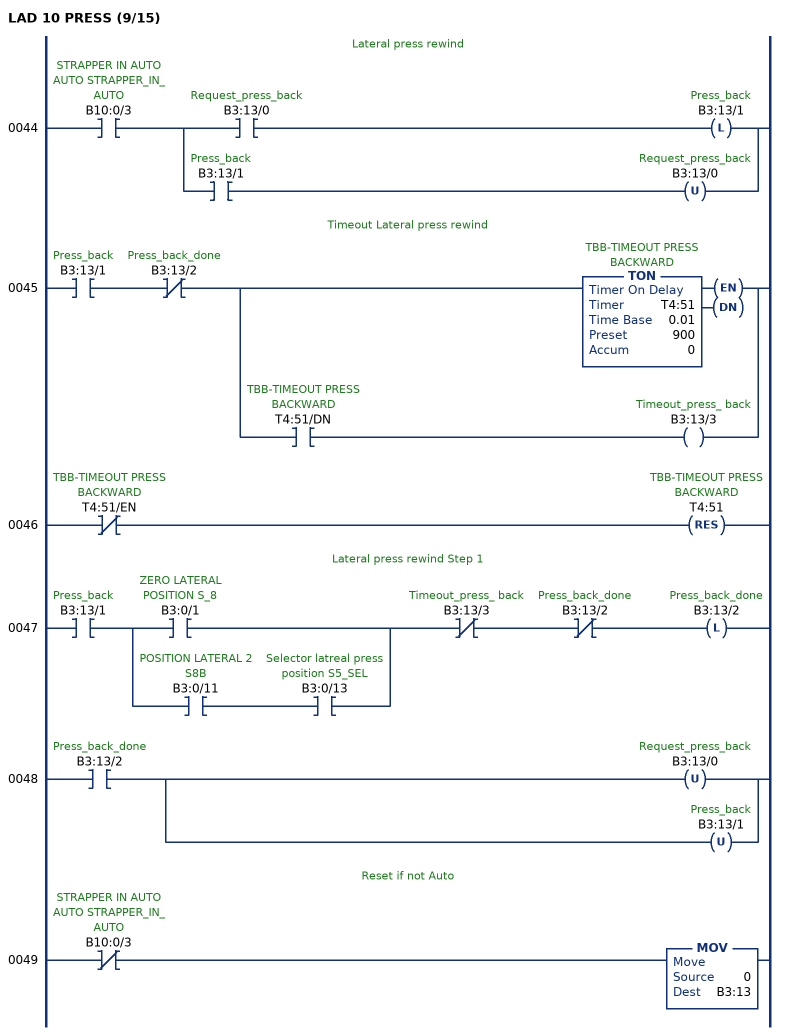
% Rung: 44 %
% Lateral press rewind %
SOR XIC B10:0/3 BST XIC B3:13/0 OTL B3:13/1 NXB XIC B3:13/1 OTU B3:13/0 BND EOR
%   B10:0/3  STRAPPER_IN_AUTO  "STRAPPER IN AUTO AUTO" %
%   B3:13/0  "Request_press_back" %
%   B3:13/1  "Press_back" %
% Rung: 45 %
% Timeout Lateral press rewind %
SOR XIC B3:13/1 XIO B3:13/2 BST TON T4:51 0.01 900 0 NXB XIC T4:51/DN OTE B3:13/3 BND EOR
%   B3:13/1  "Press_back" %
%   B3:13/2  "Press_back_done" %
%   T4:51  "TBB-TIMEOUT PRESS BACKWARD" %
%   B3:13/3  "Timeout_press_ back" %
% Rung: 46 %
SOR XIO T4:51/EN RES T4:51 EOR
%   T4:51  "TBB-TIMEOUT PRESS BACKWARD" %
% Rung: 47 %
% Lateral press rewind Step 1 %
SOR XIC B3:13/1 BST XIC B3:0/1 NXB XIC B3:0/11 XIC B3:0/13 BND XIO B3:13/3 XIO B3:13/2 OTL B3:13/2 EOR
%   B3:13/1  "Press_back" %
%   B3:0/1  S_8  "ZERO LATERAL POSITION" %
%   B3:0/11  S8B  "POSITION LATERAL 2" %
%   B3:0/13  S5_SEL  "Selector latreal press position" %
%   B3:13/3  "Timeout_press_ back" %
%   B3:13/2  "Press_back_done" %
% Rung: 48 %
SOR XIC B3:13/2 BST OTU B3:13/0 NXB OTU B3:13/1 BND EOR
%   B3:13/2  "Press_back_done" %
%   B3:13/0  "Request_press_back" %
%   B3:13/1  "Press_back" %
% Rung: 49 %
% Reset if not Auto %
SOR XIO B10:0/3 MOV 0 B3:13 EOR
%   B10:0/3  STRAPPER_IN_AUTO  "STRAPPER IN AUTO AUTO" %

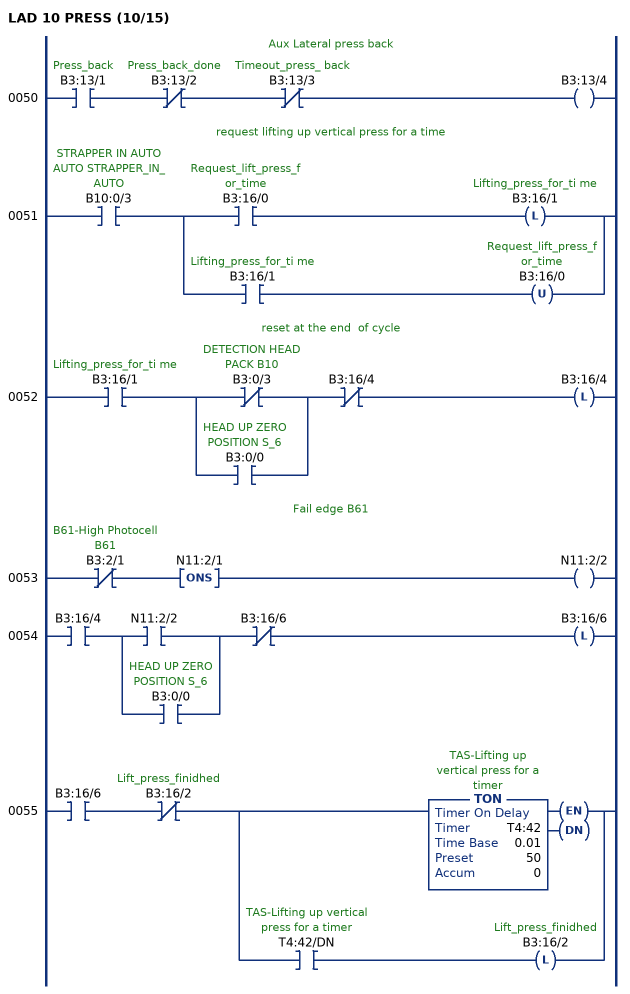
% Rung: 50 %
% Aux Lateral press back %
SOR XIC B3:13/1 XIO B3:13/2 XIO B3:13/3 OTE B3:13/4 EOR
%   B3:13/1  "Press_back" %
%   B3:13/2  "Press_back_done" %
%   B3:13/3  "Timeout_press_ back" %
% Rung: 51 %
% request lifting up vertical press for a time %
SOR XIC B10:0/3 BST XIC B3:16/0 OTL B3:16/1 NXB XIC B3:16/1 OTU B3:16/0 BND EOR
%   B10:0/3  STRAPPER_IN_AUTO  "STRAPPER IN AUTO AUTO" %
%   B3:16/0  "Request_lift_press_f or_time" %
%   B3:16/1  "Lifting_press_for_ti me" %
% Rung: 52 %
% reset at the end  of cycle %
SOR XIC B3:16/1 BST XIO B3:0/3 NXB XIC B3:0/0 BND XIO B3:16/4 OTL B3:16/4 EOR
%   B3:16/1  "Lifting_press_for_ti me" %
%   B3:0/3  B10  "DETECTION HEAD PACK" %
%   B3:0/0  S_6  "HEAD UP ZERO POSITION" %
% Rung: 53 %
% Fail edge B61 %
SOR XIO B3:2/1 ONS N11:2/1 OTE N11:2/2 EOR
%   B3:2/1  B61  "B61-High Photocell" %
% Rung: 54 %
SOR XIC B3:16/4 BST XIC N11:2/2 NXB XIC B3:0/0 BND XIO B3:16/6 OTL B3:16/6 EOR
%   B3:0/0  S_6  "HEAD UP ZERO POSITION" %
% Rung: 55 %
SOR XIC B3:16/6 XIO B3:16/2 BST TON T4:42 0.01 50 0 NXB XIC T4:42/DN OTL B3:16/2 BND EOR
%   B3:16/2  "Lift_press_finidhed" %
%   T4:42  "TAS-Lifting up vertical press for a timer" %

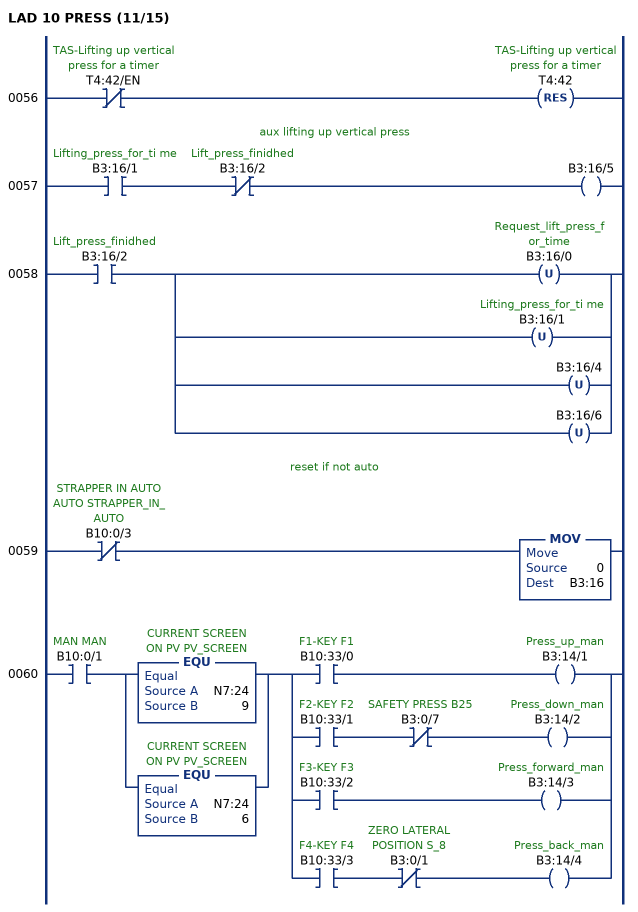
% Rung: 56 %
SOR XIO T4:42/EN RES T4:42 EOR
%   T4:42  "TAS-Lifting up vertical press for a timer" %
% Rung: 57 %
% aux lifting up vertical press %
SOR XIC B3:16/1 XIO B3:16/2 OTE B3:16/5 EOR
%   B3:16/1  "Lifting_press_for_ti me" %
%   B3:16/2  "Lift_press_finidhed" %
% Rung: 58 %
SOR XIC B3:16/2 BST OTU B3:16/0 NXB BST OTU B3:16/1 NXB BST OTU B3:16/4 NXB OTU B3:16/6 BND BND BND EOR
%   B3:16/2  "Lift_press_finidhed" %
%   B3:16/0  "Request_lift_press_f or_time" %
%   B3:16/1  "Lifting_press_for_ti me" %
% Rung: 59 %
% reset if not auto %
SOR XIO B10:0/3 MOV 0 B3:16 EOR
%   B10:0/3  STRAPPER_IN_AUTO  "STRAPPER IN AUTO AUTO" %
% Rung: 60 %
SOR XIC B10:0/1 BST EQU N7:24 9 NXB EQU N7:24 6 BND BST XIC B10:33/0 OTE B3:14/1 NXB BST XIC B10:33/1 XIO B3:0/7 OTE B3:14/2 NXB BST XIC B10:33/2 OTE B3:14/3 NXB XIC B10:33/3 XIO B3:0/1 OTE B3:14/4 BND BND BND EOR
%   B10:0/1  MAN  "MAN" %
%   N7:24  PV_SCREEN  "CURRENT SCREEN ON PV" %
%   B10:33/0  F1  "F1-KEY" %
%   B3:14/1  "Press_up_man" %
%   B10:33/1  F2  "F2-KEY" %
%   B3:0/7  B25  "SAFETY PRESS" %
%   B3:14/2  "Press_down_man" %
%   B10:33/2  F3  "F3-KEY" %
%   B3:14/3  "Press_forward_man" %
%   B10:33/3  F4  "F4-KEY" %
%   B3:0/1  S_8  "ZERO LATERAL POSITION" %
%   B3:14/4  "Press_back_man" %

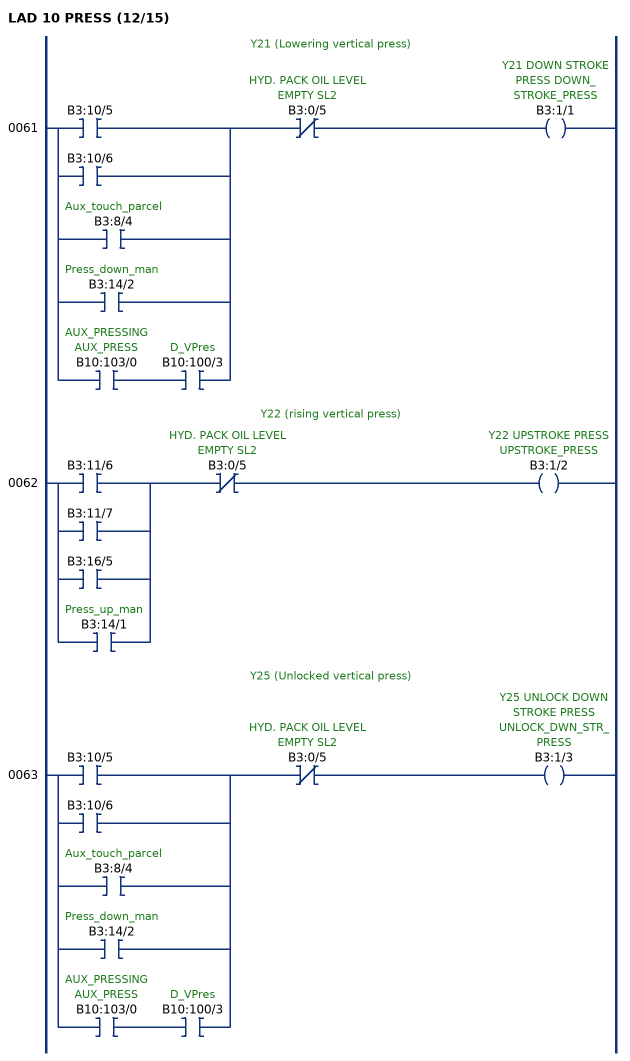
% Rung: 61 %
% Y21 (Lowering vertical press) %
SOR BST BST BST XIC B3:10/5 NXB BST XIC B3:10/6 NXB XIC B3:8/4 BND BND NXB XIC B3:14/2 BND NXB XIC B10:103/0 XIC B10:100/3 BND XIO B3:0/5 OTE B3:1/1 EOR
%   B3:8/4  "Aux_touch_parcel" %
%   B3:14/2  "Press_down_man" %
%   B10:103/0  AUX_PRESS  "AUX_PRESSING" %
%   B10:100/3  "D_VPres" %
%   B3:0/5  SL2  "HYD. PACK OIL LEVEL EMPTY" %
%   B3:1/1  DOWN_STROKE_PRESS  "Y21 DOWN STROKE PRESS" %
% Rung: 62 %
% Y22 (rising vertical press) %
SOR BST BST XIC B3:11/6 NXB BST XIC B3:11/7 NXB XIC B3:16/5 BND BND NXB XIC B3:14/1 BND XIO B3:0/5 OTE B3:1/2 EOR
%   B3:14/1  "Press_up_man" %
%   B3:0/5  SL2  "HYD. PACK OIL LEVEL EMPTY" %
%   B3:1/2  UPSTROKE_PRESS  "Y22 UPSTROKE PRESS" %
% Rung: 63 %
% Y25 (Unlocked vertical press) %
SOR BST XIC B3:10/5 NXB BST BST XIC B3:10/6 NXB XIC B3:8/4 BND NXB BST XIC B3:14/2 NXB XIC B10:103/0 XIC B10:100/3 BND BND BND XIO B3:0/5 OTE B3:1/3 EOR
%   B3:8/4  "Aux_touch_parcel" %
%   B3:14/2  "Press_down_man" %
%   B10:103/0  AUX_PRESS  "AUX_PRESSING" %
%   B10:100/3  "D_VPres" %
%   B3:0/5  SL2  "HYD. PACK OIL LEVEL EMPTY" %
%   B3:1/3  UNLOCK_DWN_STR_PRESS  "Y25 UNLOCK DOWN STROKE PRESS" %

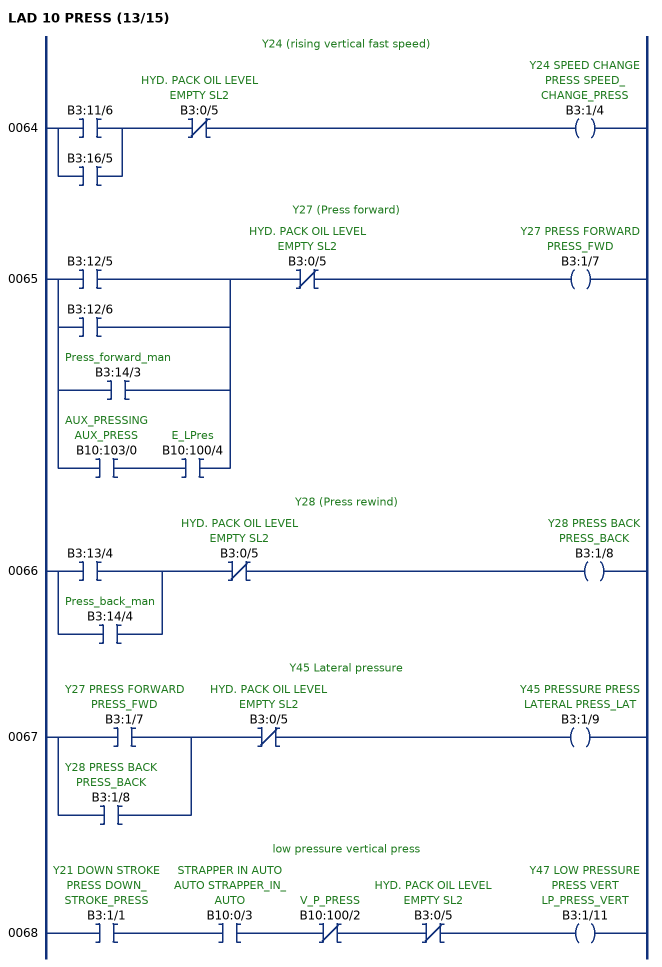
% Rung: 64 %
% Y24 (rising vertical fast speed) %
SOR BST XIC B3:11/6 NXB XIC B3:16/5 BND XIO B3:0/5 OTE B3:1/4 EOR
%   B3:0/5  SL2  "HYD. PACK OIL LEVEL EMPTY" %
%   B3:1/4  SPEED_CHANGE_PRESS  "Y24 SPEED CHANGE PRESS" %
% Rung: 65 %
% Y27 (Press forward) %
SOR BST XIC B3:12/5 NXB BST XIC B3:12/6 NXB BST XIC B3:14/3 NXB XIC B10:103/0 XIC B10:100/4 BND BND BND XIO B3:0/5 OTE B3:1/7 EOR
%   B3:14/3  "Press_forward_man" %
%   B10:103/0  AUX_PRESS  "AUX_PRESSING" %
%   B10:100/4  "E_LPres" %
%   B3:0/5  SL2  "HYD. PACK OIL LEVEL EMPTY" %
%   B3:1/7  PRESS_FWD  "Y27 PRESS FORWARD" %
% Rung: 66 %
% Y28 (Press rewind) %
SOR BST XIC B3:13/4 NXB XIC B3:14/4 BND XIO B3:0/5 OTE B3:1/8 EOR
%   B3:14/4  "Press_back_man" %
%   B3:0/5  SL2  "HYD. PACK OIL LEVEL EMPTY" %
%   B3:1/8  PRESS_BACK  "Y28 PRESS BACK" %
% Rung: 67 %
% Y45 Lateral pressure %
SOR BST XIC B3:1/7 NXB XIC B3:1/8 BND XIO B3:0/5 OTE B3:1/9 EOR
%   B3:1/7  PRESS_FWD  "Y27 PRESS FORWARD" %
%   B3:1/8  PRESS_BACK  "Y28 PRESS BACK" %
%   B3:0/5  SL2  "HYD. PACK OIL LEVEL EMPTY" %
%   B3:1/9  PRESS_LAT  "Y45 PRESSURE PRESS LATERAL" %
% Rung: 68 %
% low pressure vertical press %
SOR XIC B3:1/1 XIC B10:0/3 XIO B10:100/2 XIO B3:0/5 OTE B3:1/11 EOR
%   B3:1/1  DOWN_STROKE_PRESS  "Y21 DOWN STROKE PRESS" %
%   B10:0/3  STRAPPER_IN_AUTO  "STRAPPER IN AUTO AUTO" %
%   B10:100/2  "V_P_PRESS" %
%   B3:0/5  SL2  "HYD. PACK OIL LEVEL EMPTY" %
%   B3:1/11  LP_PRESS_VERT  "Y47 LOW PRESSURE PRESS VERT" %

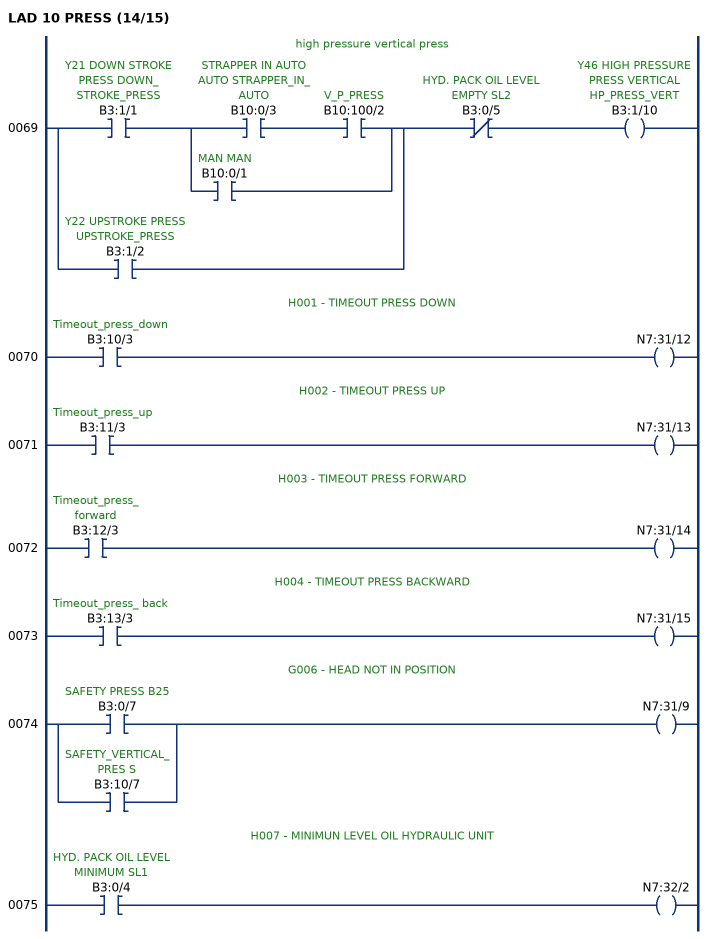
% Rung: 69 %
% high pressure vertical press %
SOR BST XIC B3:1/1 BST XIC B10:0/3 XIC B10:100/2 NXB XIC B10:0/1 BND NXB XIC B3:1/2 BND XIO B3:0/5 OTE B3:1/10 EOR
%   B3:1/1  DOWN_STROKE_PRESS  "Y21 DOWN STROKE PRESS" %
%   B10:0/3  STRAPPER_IN_AUTO  "STRAPPER IN AUTO AUTO" %
%   B10:100/2  "V_P_PRESS" %
%   B10:0/1  MAN  "MAN" %
%   B3:1/2  UPSTROKE_PRESS  "Y22 UPSTROKE PRESS" %
%   B3:0/5  SL2  "HYD. PACK OIL LEVEL EMPTY" %
%   B3:1/10  HP_PRESS_VERT  "Y46 HIGH PRESSURE PRESS VERTICAL" %
% Rung: 70 %
% H001 - TIMEOUT PRESS DOWN %
SOR XIC B3:10/3 OTE N7:31/12 EOR
%   B3:10/3  "Timeout_press_down" %
% Rung: 71 %
% H002 - TIMEOUT PRESS UP %
SOR XIC B3:11/3 OTE N7:31/13 EOR
%   B3:11/3  "Timeout_press_up" %
% Rung: 72 %
% H003 - TIMEOUT PRESS FORWARD %
SOR XIC B3:12/3 OTE N7:31/14 EOR
%   B3:12/3  "Timeout_press_ forward" %
% Rung: 73 %
% H004 - TIMEOUT PRESS BACKWARD %
SOR XIC B3:13/3 OTE N7:31/15 EOR
%   B3:13/3  "Timeout_press_ back" %
% Rung: 74 %
% G006 - HEAD NOT IN POSITION %
SOR BST XIC B3:0/7 NXB XIC B3:10/7 BND OTE N7:31/9 EOR
%   B3:0/7  B25  "SAFETY PRESS" %
%   B3:10/7  "SAFETY_VERTICAL_PRES S" %
% Rung: 75 %
% H007 - MINIMUN LEVEL OIL HYDRAULIC UNIT %
SOR XIC B3:0/4 OTE N7:32/2 EOR
%   B3:0/4  SL1  "HYD. PACK OIL LEVEL MINIMUM" %

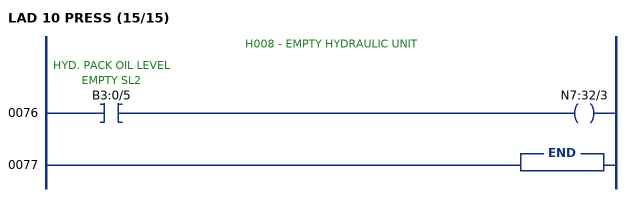
% Rung: 76 %
% H008 - EMPTY HYDRAULIC UNIT %
SOR XIC B3:0/5 OTE N7:32/3 EOR
%   B3:0/5  SL2  "HYD. PACK OIL LEVEL EMPTY" %
% Rung: 77 %
SOR END EOR

LADDER 11 "PUSH_BUNK"
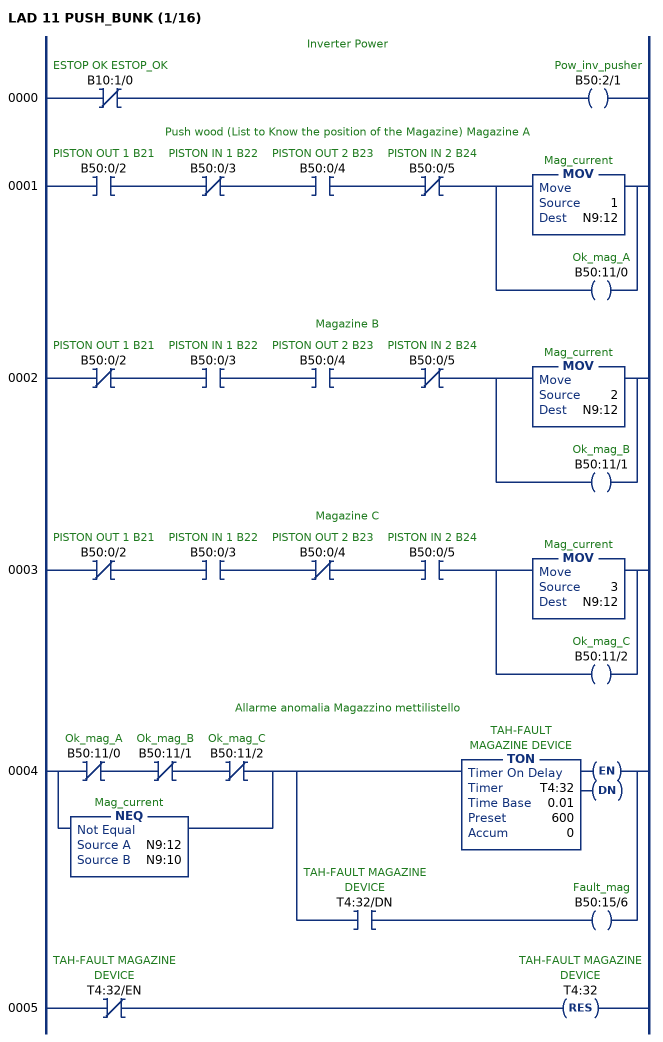
% Rung: 0 %
% Inverter Power %
SOR XIO B10:1/0 OTE B50:2/1 EOR
%   B10:1/0  ESTOP_OK  "ESTOP OK" %
%   B50:2/1  "Pow_inv_pusher" %
% Rung: 1 %
% Push wood (List to Know the position of the Magazine) Magazine A %
SOR XIC B50:0/2 XIO B50:0/3 XIC B50:0/4 XIO B50:0/5 BST MOV 1 N9:12 NXB OTE B50:11/0 BND EOR
%   B50:0/2  B21  "PISTON OUT 1" %
%   B50:0/3  B22  "PISTON IN 1" %
%   B50:0/4  B23  "PISTON OUT 2" %
%   B50:0/5  B24  "PISTON IN 2" %
%   N9:12  "Mag_current" %
%   B50:11/0  "Ok_mag_A" %
% Rung: 2 %
% Magazine B %
SOR XIO B50:0/2 XIC B50:0/3 XIC B50:0/4 XIO B50:0/5 BST MOV 2 N9:12 NXB OTE B50:11/1 BND EOR
%   B50:0/2  B21  "PISTON OUT 1" %
%   B50:0/3  B22  "PISTON IN 1" %
%   B50:0/4  B23  "PISTON OUT 2" %
%   B50:0/5  B24  "PISTON IN 2" %
%   N9:12  "Mag_current" %
%   B50:11/1  "Ok_mag_B" %
% Rung: 3 %
% Magazine C %
SOR XIO B50:0/2 XIC B50:0/3 XIO B50:0/4 XIC B50:0/5 BST MOV 3 N9:12 NXB OTE B50:11/2 BND EOR
%   B50:0/2  B21  "PISTON OUT 1" %
%   B50:0/3  B22  "PISTON IN 1" %
%   B50:0/4  B23  "PISTON OUT 2" %
%   B50:0/5  B24  "PISTON IN 2" %
%   N9:12  "Mag_current" %
%   B50:11/2  "Ok_mag_C" %
% Rung: 4 %
% Allarme anomalia Magazzino mettilistello %
SOR BST XIO B50:11/0 XIO B50:11/1 XIO B50:11/2 NXB NEQ N9:12 N9:10 BND BST TON T4:32 0.01 600 0 NXB XIC T4:32/DN OTE B50:15/6 BND EOR
%   B50:11/0  "Ok_mag_A" %
%   B50:11/1  "Ok_mag_B" %
%   B50:11/2  "Ok_mag_C" %
%   N9:12  "Mag_current" %
%   N9:10  "Mag_request" %
%   T4:32  "TAH-FAULT MAGAZINE DEVICE" %
%   B50:15/6  "Fault_mag" %
% Rung: 5 %
SOR XIO T4:32/EN RES T4:32 EOR
%   T4:32  "TAH-FAULT MAGAZINE DEVICE" %

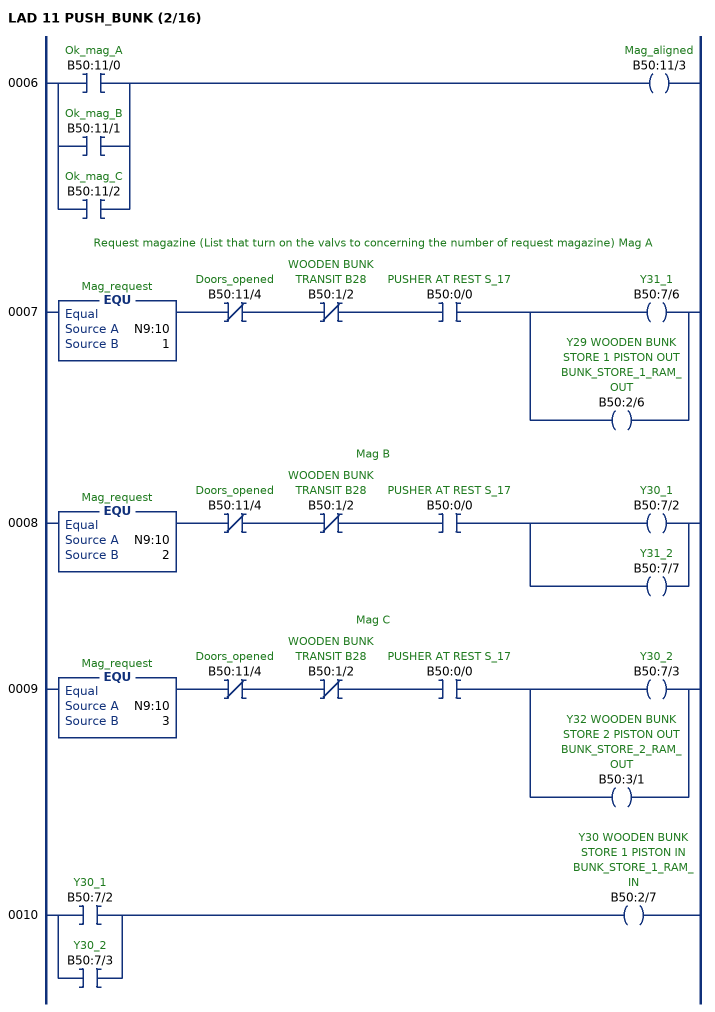
% Rung: 6 %
SOR BST XIC B50:11/0 NXB BST XIC B50:11/1 NXB XIC B50:11/2 BND BND OTE B50:11/3 EOR
%   B50:11/0  "Ok_mag_A" %
%   B50:11/1  "Ok_mag_B" %
%   B50:11/2  "Ok_mag_C" %
%   B50:11/3  "Mag_aligned" %
% Rung: 7 %
% Request magazine (List that turn on the valvs to concerning the number of request magazine) Mag A %
SOR EQU N9:10 1 XIO B50:11/4 XIO B50:1/2 XIC B50:0/0 BST OTE B50:7/6 NXB OTE B50:2/6 BND EOR
%   N9:10  "Mag_request" %
%   B50:11/4  "Doors_opened" %
%   B50:1/2  B28  "WOODEN BUNK TRANSIT" %
%   B50:0/0  S_17  "PUSHER AT REST" %
%   B50:7/6  "Y31_1" %
%   B50:2/6  BUNK_STORE_1_RAM_OUT  "Y29 WOODEN BUNK STORE 1 PISTON OUT" %
% Rung: 8 %
% Mag B %
SOR EQU N9:10 2 XIO B50:11/4 XIO B50:1/2 XIC B50:0/0 BST OTE B50:7/2 NXB OTE B50:7/7 BND EOR
%   N9:10  "Mag_request" %
%   B50:11/4  "Doors_opened" %
%   B50:1/2  B28  "WOODEN BUNK TRANSIT" %
%   B50:0/0  S_17  "PUSHER AT REST" %
%   B50:7/2  "Y30_1" %
%   B50:7/7  "Y31_2" %
% Rung: 9 %
% Mag C %
SOR EQU N9:10 3 XIO B50:11/4 XIO B50:1/2 XIC B50:0/0 BST OTE B50:7/3 NXB OTE B50:3/1 BND EOR
%   N9:10  "Mag_request" %
%   B50:11/4  "Doors_opened" %
%   B50:1/2  B28  "WOODEN BUNK TRANSIT" %
%   B50:0/0  S_17  "PUSHER AT REST" %
%   B50:7/3  "Y30_2" %
%   B50:3/1  BUNK_STORE_2_RAM_OUT  "Y32 WOODEN BUNK STORE 2 PISTON OUT" %
% Rung: 10 %
SOR BST XIC B50:7/2 NXB XIC B50:7/3 BND OTE B50:2/7 EOR
%   B50:7/2  "Y30_1" %
%   B50:7/3  "Y30_2" %
%   B50:2/7  BUNK_STORE_1_RAM_IN  "Y30 WOODEN BUNK STORE 1 PISTON IN" %

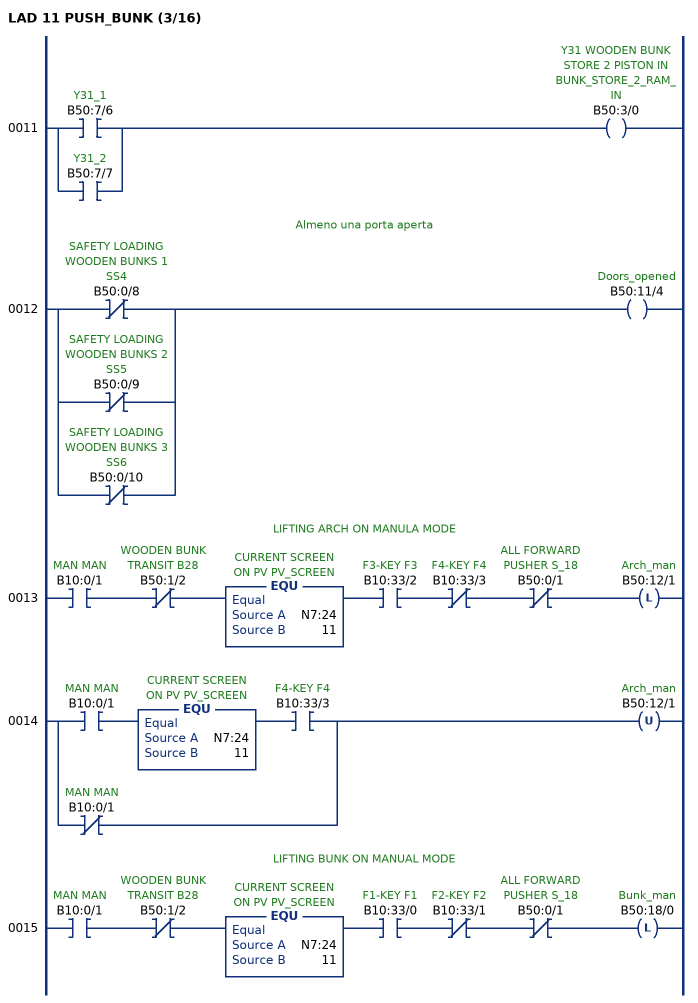
% Rung: 11 %
SOR BST XIC B50:7/6 NXB XIC B50:7/7 BND OTE B50:3/0 EOR
%   B50:7/6  "Y31_1" %
%   B50:7/7  "Y31_2" %
%   B50:3/0  BUNK_STORE_2_RAM_IN  "Y31 WOODEN BUNK STORE 2 PISTON IN" %
% Rung: 12 %
% Almeno una porta aperta %
SOR BST XIO B50:0/8 NXB BST XIO B50:0/9 NXB XIO B50:0/10 BND BND OTE B50:11/4 EOR
%   B50:0/8  SS4  "SAFETY LOADING WOODEN BUNKS 1" %
%   B50:0/9  SS5  "SAFETY LOADING WOODEN BUNKS 2" %
%   B50:0/10  SS6  "SAFETY LOADING WOODEN BUNKS 3" %
%   B50:11/4  "Doors_opened" %
% Rung: 13 %
% LIFTING ARCH ON MANULA MODE %
SOR XIC B10:0/1 XIO B50:1/2 EQU N7:24 11 XIC B10:33/2 XIO B10:33/3 XIO B50:0/1 OTL B50:12/1 EOR
%   B10:0/1  MAN  "MAN" %
%   B50:1/2  B28  "WOODEN BUNK TRANSIT" %
%   N7:24  PV_SCREEN  "CURRENT SCREEN ON PV" %
%   B10:33/2  F3  "F3-KEY" %
%   B10:33/3  F4  "F4-KEY" %
%   B50:0/1  S_18  "ALL FORWARD PUSHER" %
%   B50:12/1  "Arch_man" %
% Rung: 14 %
SOR BST XIC B10:0/1 EQU N7:24 11 XIC B10:33/3 NXB XIO B10:0/1 BND OTU B50:12/1 EOR
%   B10:0/1  MAN  "MAN" %
%   N7:24  PV_SCREEN  "CURRENT SCREEN ON PV" %
%   B10:33/3  F4  "F4-KEY" %
%   B50:12/1  "Arch_man" %
% Rung: 15 %
% LIFTING BUNK ON MANUAL MODE %
SOR XIC B10:0/1 XIO B50:1/2 EQU N7:24 11 XIC B10:33/0 XIO B10:33/1 XIO B50:0/1 OTL B50:18/0 EOR
%   B10:0/1  MAN  "MAN" %
%   B50:1/2  B28  "WOODEN BUNK TRANSIT" %
%   N7:24  PV_SCREEN  "CURRENT SCREEN ON PV" %
%   B10:33/0  F1  "F1-KEY" %
%   B10:33/1  F2  "F2-KEY" %
%   B50:0/1  S_18  "ALL FORWARD PUSHER" %
%   B50:18/0  "Bunk_man" %

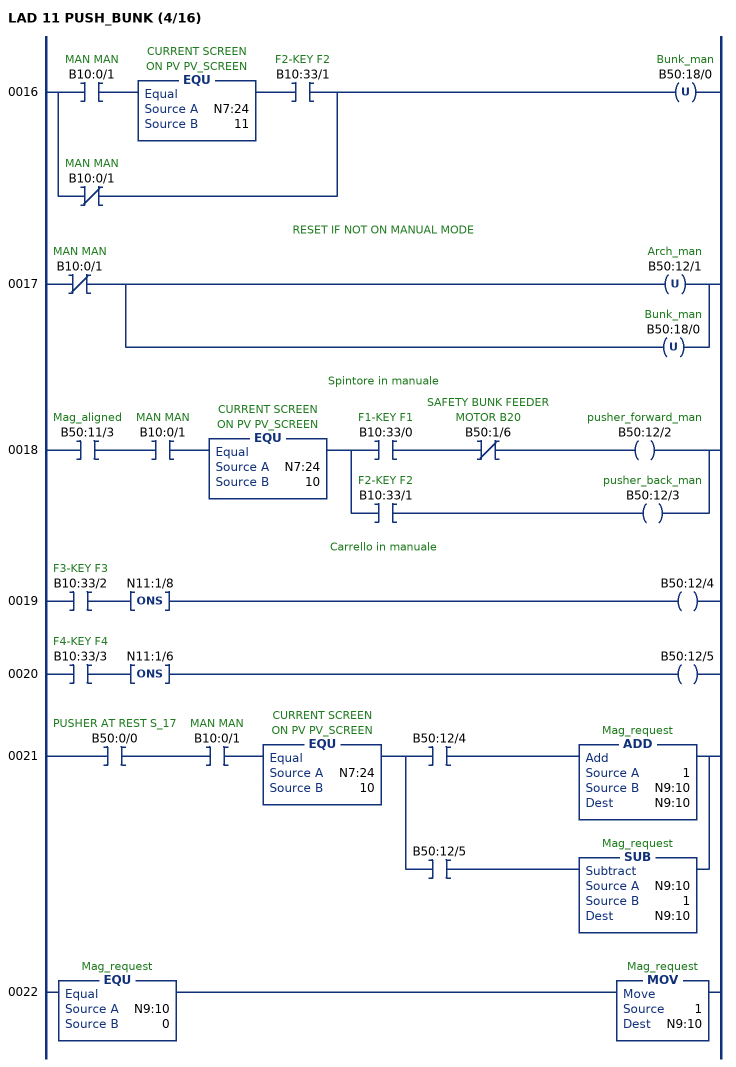
% Rung: 16 %
SOR BST XIC B10:0/1 EQU N7:24 11 XIC B10:33/1 NXB XIO B10:0/1 BND OTU B50:18/0 EOR
%   B10:0/1  MAN  "MAN" %
%   N7:24  PV_SCREEN  "CURRENT SCREEN ON PV" %
%   B10:33/1  F2  "F2-KEY" %
%   B50:18/0  "Bunk_man" %
% Rung: 17 %
% RESET IF NOT ON MANUAL MODE %
SOR XIO B10:0/1 BST OTU B50:12/1 NXB OTU B50:18/0 BND EOR
%   B10:0/1  MAN  "MAN" %
%   B50:12/1  "Arch_man" %
%   B50:18/0  "Bunk_man" %
% Rung: 18 %
% Spintore in manuale %
SOR XIC B50:11/3 XIC B10:0/1 EQU N7:24 10 BST XIC B10:33/0 XIO B50:1/6 OTE B50:12/2 NXB XIC B10:33/1 OTE B50:12/3 BND EOR
%   B50:11/3  "Mag_aligned" %
%   B10:0/1  MAN  "MAN" %
%   N7:24  PV_SCREEN  "CURRENT SCREEN ON PV" %
%   B10:33/0  F1  "F1-KEY" %
%   B50:1/6  B20  "SAFETY BUNK FEEDER MOTOR" %
%   B50:12/2  "pusher_forward_man" %
%   B10:33/1  F2  "F2-KEY" %
%   B50:12/3  "pusher_back_man" %
% Rung: 19 %
% Carrello in manuale %
SOR XIC B10:33/2 ONS N11:1/8 OTE B50:12/4 EOR
%   B10:33/2  F3  "F3-KEY" %
% Rung: 20 %
SOR XIC B10:33/3 ONS N11:1/6 OTE B50:12/5 EOR
%   B10:33/3  F4  "F4-KEY" %
% Rung: 21 %
SOR XIC B50:0/0 XIC B10:0/1 EQU N7:24 10 BST XIC B50:12/4 ADD 1 N9:10 N9:10 NXB XIC B50:12/5 SUB N9:10 1 N9:10 BND EOR
%   B50:0/0  S_17  "PUSHER AT REST" %
%   B10:0/1  MAN  "MAN" %
%   N7:24  PV_SCREEN  "CURRENT SCREEN ON PV" %
%   N9:10  "Mag_request" %
% Rung: 22 %
SOR EQU N9:10 0 MOV 1 N9:10 EOR
%   N9:10  "Mag_request" %

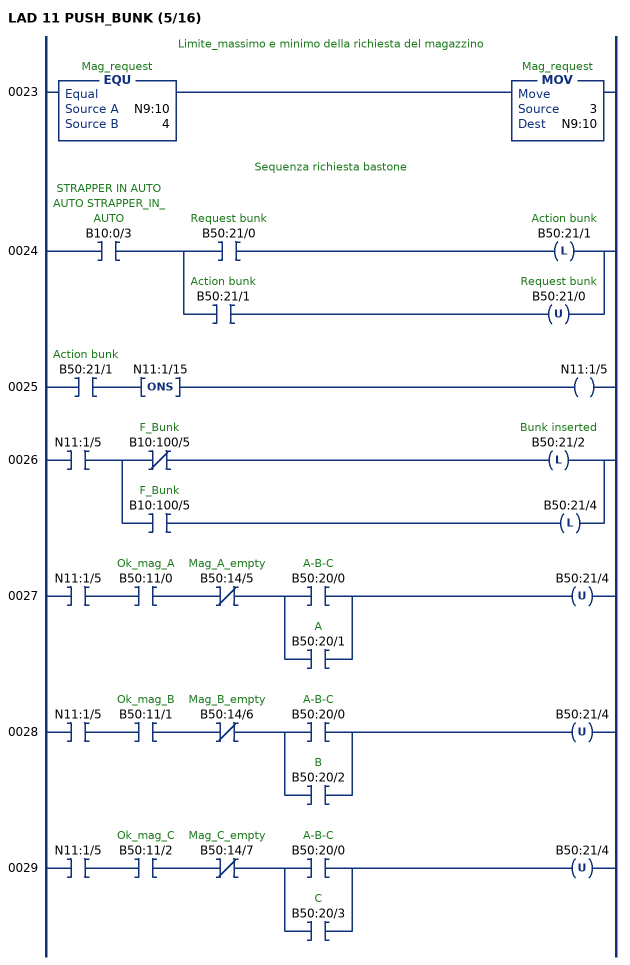
% Rung: 23 %
% Limite_massimo e minimo della richiesta del magazzino %
SOR EQU N9:10 4 MOV 3 N9:10 EOR
%   N9:10  "Mag_request" %
% Rung: 24 %
% Sequenza richiesta bastone %
SOR XIC B10:0/3 BST XIC B50:21/0 OTL B50:21/1 NXB XIC B50:21/1 OTU B50:21/0 BND EOR
%   B10:0/3  STRAPPER_IN_AUTO  "STRAPPER IN AUTO AUTO" %
%   B50:21/0  "Request bunk" %
%   B50:21/1  "Action bunk" %
% Rung: 25 %
SOR XIC B50:21/1 ONS N11:1/15 OTE N11:1/5 EOR
%   B50:21/1  "Action bunk" %
% Rung: 26 %
SOR XIC N11:1/5 BST XIO B10:100/5 OTL B50:21/2 NXB XIC B10:100/5 OTL B50:21/4 BND EOR
%   B10:100/5  "F_Bunk" %
%   B50:21/2  "Bunk inserted" %
% Rung: 27 %
SOR XIC N11:1/5 XIC B50:11/0 XIO B50:14/5 BST XIC B50:20/0 NXB XIC B50:20/1 BND OTU B50:21/4 EOR
%   B50:11/0  "Ok_mag_A" %
%   B50:14/5  "Mag_A_empty" %
%   B50:20/0  "A-B-C" %
%   B50:20/1  "A" %
% Rung: 28 %
SOR XIC N11:1/5 XIC B50:11/1 XIO B50:14/6 BST XIC B50:20/0 NXB XIC B50:20/2 BND OTU B50:21/4 EOR
%   B50:11/1  "Ok_mag_B" %
%   B50:14/6  "Mag_B_empty" %
%   B50:20/0  "A-B-C" %
%   B50:20/2  "B" %
% Rung: 29 %
SOR XIC N11:1/5 XIC B50:11/2 XIO B50:14/7 BST XIC B50:20/0 NXB XIC B50:20/3 BND OTU B50:21/4 EOR
%   B50:11/2  "Ok_mag_C" %
%   B50:14/7  "Mag_C_empty" %
%   B50:20/0  "A-B-C" %
%   B50:20/3  "C" %

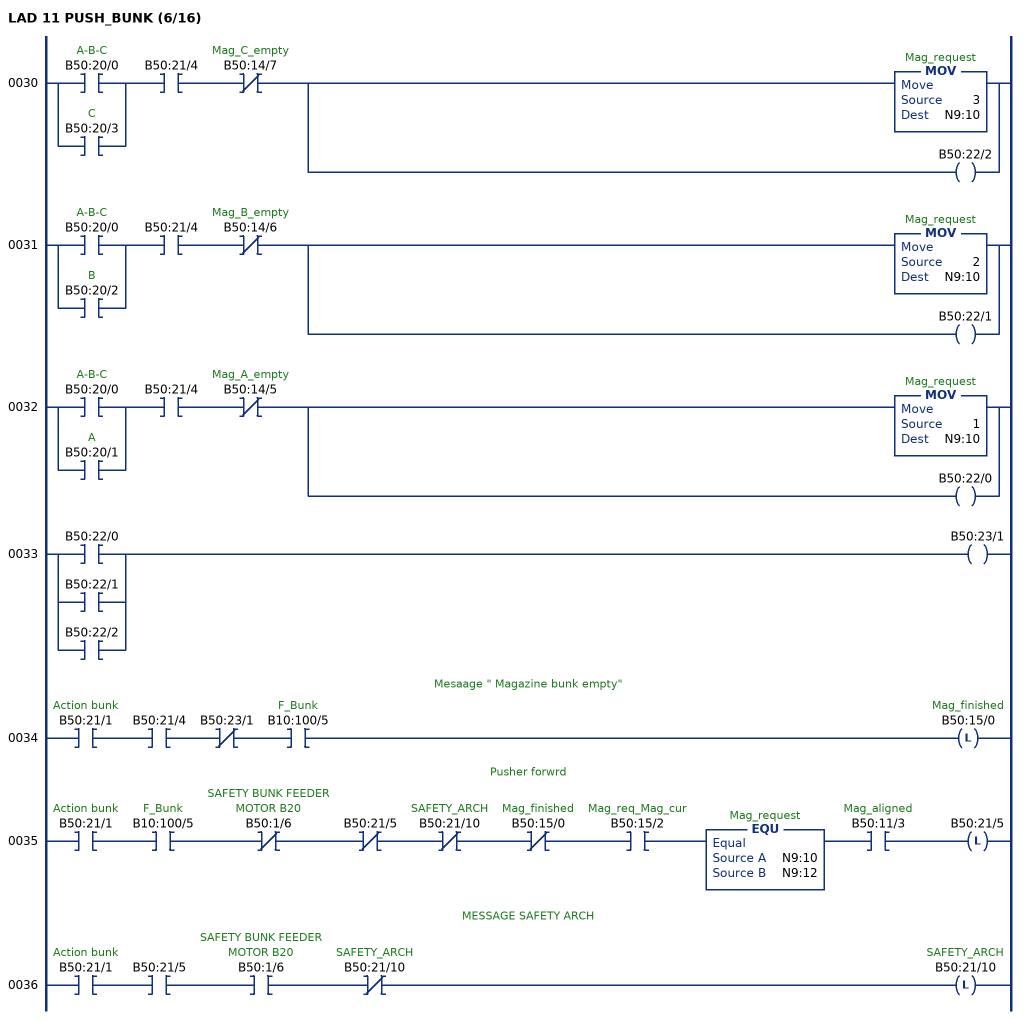
% Rung: 30 %
SOR BST XIC B50:20/0 NXB XIC B50:20/3 BND XIC B50:21/4 XIO B50:14/7 BST MOV 3 N9:10 NXB OTE B50:22/2 BND EOR
%   B50:20/0  "A-B-C" %
%   B50:20/3  "C" %
%   B50:14/7  "Mag_C_empty" %
%   N9:10  "Mag_request" %
% Rung: 31 %
SOR BST XIC B50:20/0 NXB XIC B50:20/2 BND XIC B50:21/4 XIO B50:14/6 BST MOV 2 N9:10 NXB OTE B50:22/1 BND EOR
%   B50:20/0  "A-B-C" %
%   B50:20/2  "B" %
%   B50:14/6  "Mag_B_empty" %
%   N9:10  "Mag_request" %
% Rung: 32 %
SOR BST XIC B50:20/0 NXB XIC B50:20/1 BND XIC B50:21/4 XIO B50:14/5 BST MOV 1 N9:10 NXB OTE B50:22/0 BND EOR
%   B50:20/0  "A-B-C" %
%   B50:20/1  "A" %
%   B50:14/5  "Mag_A_empty" %
%   N9:10  "Mag_request" %
% Rung: 33 %
SOR BST XIC B50:22/0 NXB BST XIC B50:22/1 NXB XIC B50:22/2 BND BND OTE B50:23/1 EOR
% Rung: 34 %
% Mesaage " Magazine bunk empty" %
SOR XIC B50:21/1 XIC B50:21/4 XIO B50:23/1 XIC B10:100/5 OTL B50:15/0 EOR
%   B50:21/1  "Action bunk" %
%   B10:100/5  "F_Bunk" %
%   B50:15/0  "Mag_finished" %
% Rung: 35 %
% Pusher forwrd %
SOR XIC B50:21/1 XIC B10:100/5 XIO B50:1/6 XIO B50:21/5 XIO B50:21/10 XIO B50:15/0 XIC B50:15/2 EQU N9:10 N9:12 XIC B50:11/3 OTL B50:21/5 EOR
%   B50:21/1  "Action bunk" %
%   B10:100/5  "F_Bunk" %
%   B50:1/6  B20  "SAFETY BUNK FEEDER MOTOR" %
%   B50:21/10  "SAFETY_ARCH" %
%   B50:15/0  "Mag_finished" %
%   B50:15/2  "Mag_req_Mag_cur" %
%   N9:10  "Mag_request" %
%   N9:12  "Mag_current" %
%   B50:11/3  "Mag_aligned" %
% Rung: 36 %
% MESSAGE SAFETY ARCH %
SOR XIC B50:21/1 XIC B50:21/5 XIC B50:1/6 XIO B50:21/10 OTL B50:21/10 EOR
%   B50:21/1  "Action bunk" %
%   B50:1/6  B20  "SAFETY BUNK FEEDER MOTOR" %
%   B50:21/10  "SAFETY_ARCH" %

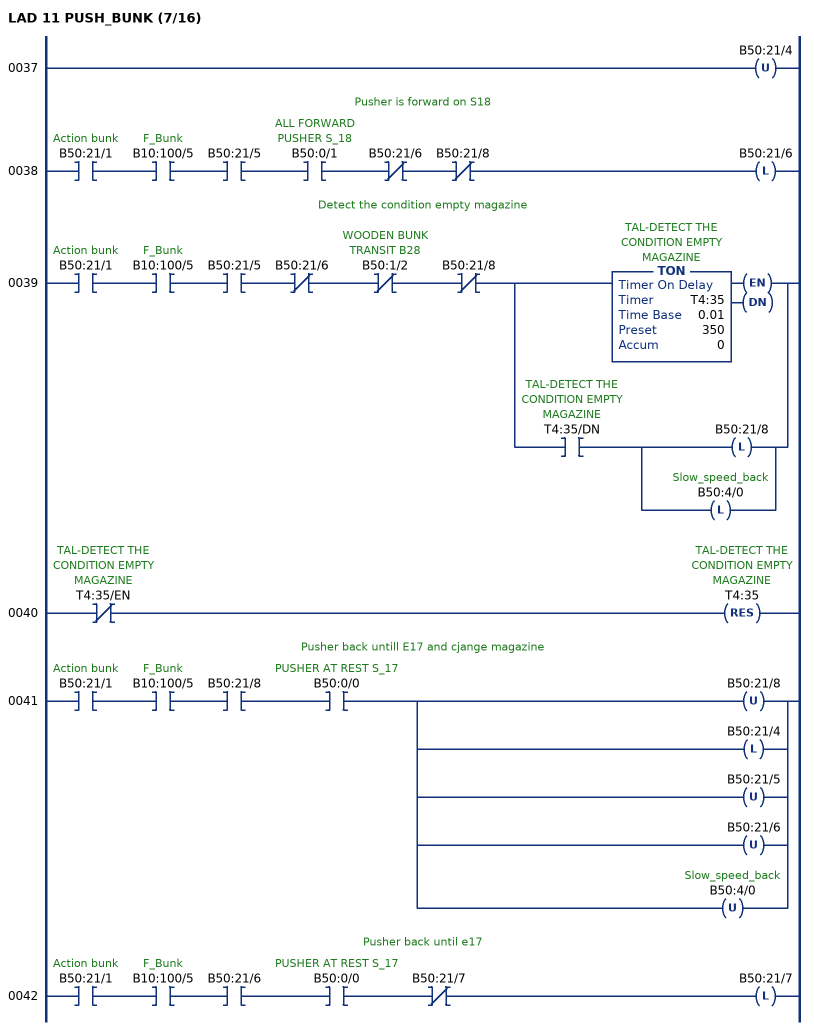
% Rung: 37 %
SOR OTU B50:21/4 EOR
% Rung: 38 %
% Pusher is forward on S18 %
SOR XIC B50:21/1 XIC B10:100/5 XIC B50:21/5 XIC B50:0/1 XIO B50:21/6 XIO B50:21/8 OTL B50:21/6 EOR
%   B50:21/1  "Action bunk" %
%   B10:100/5  "F_Bunk" %
%   B50:0/1  S_18  "ALL FORWARD PUSHER" %
% Rung: 39 %
% Detect the condition empty magazine %
SOR XIC B50:21/1 XIC B10:100/5 XIC B50:21/5 XIO B50:21/6 XIO B50:1/2 XIO B50:21/8 BST TON T4:35 0.01 350 0 NXB XIC T4:35/DN BST OTL B50:21/8 NXB OTL B50:4/0 BND BND EOR
%   B50:21/1  "Action bunk" %
%   B10:100/5  "F_Bunk" %
%   B50:1/2  B28  "WOODEN BUNK TRANSIT" %
%   T4:35  "TAL-DETECT THE CONDITION EMPTY MAGAZINE" %
%   B50:4/0  "Slow_speed_back" %
% Rung: 40 %
SOR XIO T4:35/EN RES T4:35 EOR
%   T4:35  "TAL-DETECT THE CONDITION EMPTY MAGAZINE" %
% Rung: 41 %
% Pusher back untill E17 and cjange magazine %
SOR XIC B50:21/1 XIC B10:100/5 XIC B50:21/8 XIC B50:0/0 BST OTU B50:21/8 NXB BST OTL B50:21/4 NXB BST OTU B50:21/5 NXB BST OTU B50:21/6 NXB OTU B50:4/0 BND BND BND BND EOR
%   B50:21/1  "Action bunk" %
%   B10:100/5  "F_Bunk" %
%   B50:0/0  S_17  "PUSHER AT REST" %
%   B50:4/0  "Slow_speed_back" %
% Rung: 42 %
% Pusher back until e17 %
SOR XIC B50:21/1 XIC B10:100/5 XIC B50:21/6 XIC B50:0/0 XIO B50:21/7 OTL B50:21/7 EOR
%   B50:21/1  "Action bunk" %
%   B10:100/5  "F_Bunk" %
%   B50:0/0  S_17  "PUSHER AT REST" %

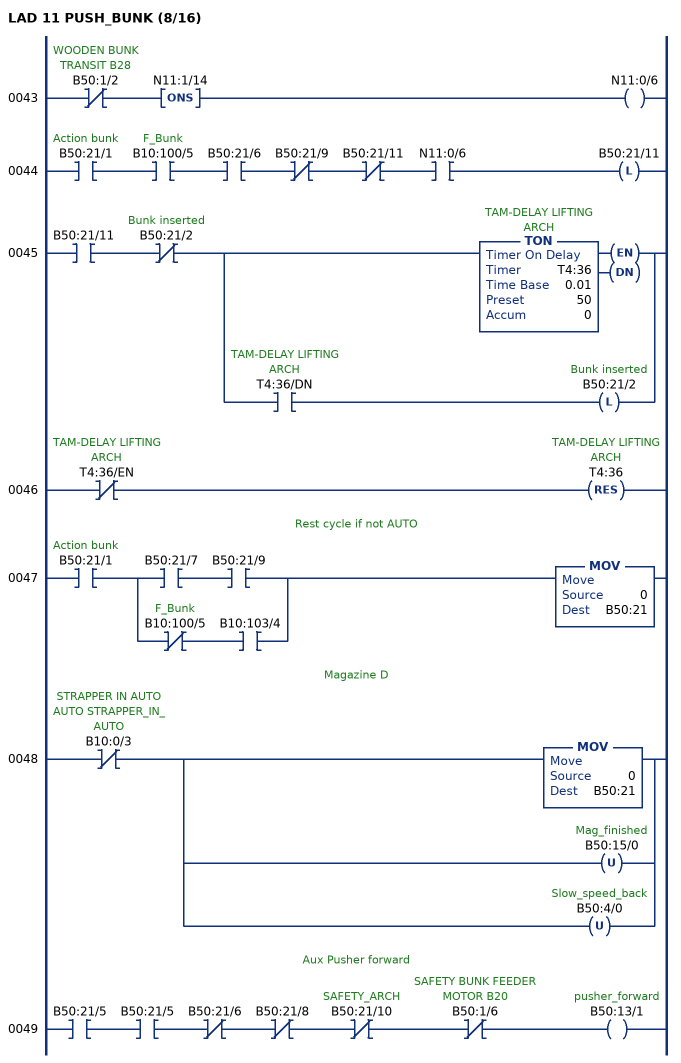
% Rung: 43 %
SOR XIO B50:1/2 ONS N11:1/14 OTE N11:0/6 EOR
%   B50:1/2  B28  "WOODEN BUNK TRANSIT" %
% Rung: 44 %
SOR XIC B50:21/1 XIC B10:100/5 XIC B50:21/6 XIO B50:21/9 XIO B50:21/11 XIC N11:0/6 OTL B50:21/11 EOR
%   B50:21/1  "Action bunk" %
%   B10:100/5  "F_Bunk" %
% Rung: 45 %
SOR XIC B50:21/11 XIO B50:21/2 BST TON T4:36 0.01 50 0 NXB XIC T4:36/DN OTL B50:21/2 BND EOR
%   B50:21/2  "Bunk inserted" %
%   T4:36  "TAM-DELAY LIFTING ARCH" %
% Rung: 46 %
SOR XIO T4:36/EN RES T4:36 EOR
%   T4:36  "TAM-DELAY LIFTING ARCH" %
% Rung: 47 %
% Rest cycle if not AUTO %
SOR XIC B50:21/1 BST XIC B50:21/7 XIC B50:21/9 NXB XIO B10:100/5 XIC B10:103/4 BND MOV 0 B50:21 EOR
%   B50:21/1  "Action bunk" %
%   B10:100/5  "F_Bunk" %
% Rung: 48 %
% Magazine D %
SOR XIO B10:0/3 BST MOV 0 B50:21 NXB BST OTU B50:15/0 NXB OTU B50:4/0 BND BND EOR
%   B10:0/3  STRAPPER_IN_AUTO  "STRAPPER IN AUTO AUTO" %
%   B50:15/0  "Mag_finished" %
%   B50:4/0  "Slow_speed_back" %
% Rung: 49 %
% Aux Pusher forward %
SOR XIC B50:21/5 XIC B50:21/5 XIO B50:21/6 XIO B50:21/8 XIO B50:21/10 XIO B50:1/6 OTE B50:13/1 EOR
%   B50:21/10  "SAFETY_ARCH" %
%   B50:1/6  B20  "SAFETY BUNK FEEDER MOTOR" %
%   B50:13/1  "pusher_forward" %

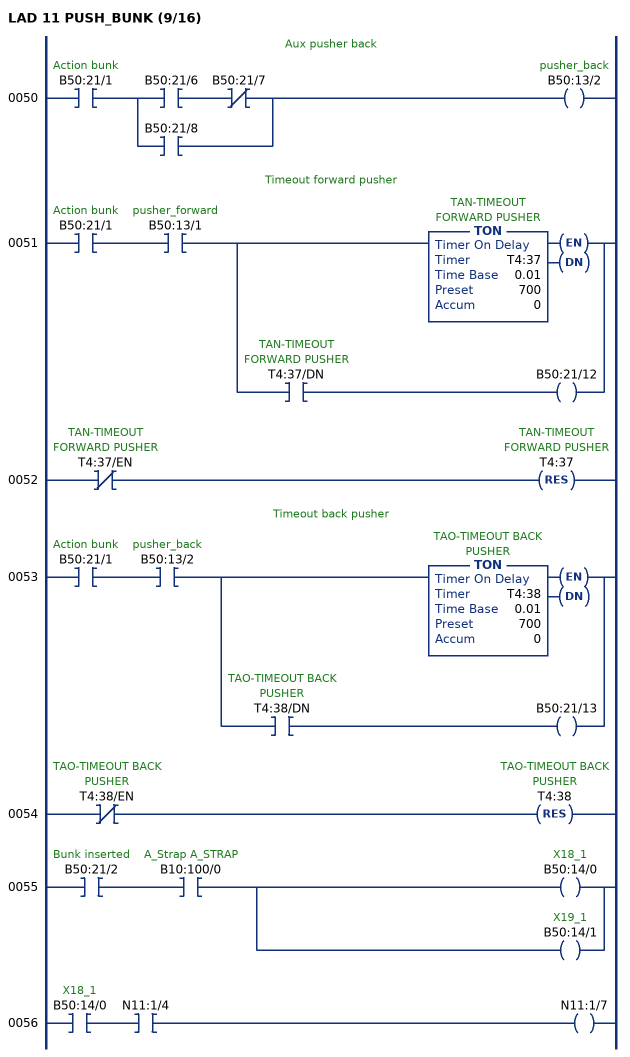
% Rung: 50 %
% Aux pusher back %
SOR XIC B50:21/1 BST XIC B50:21/6 XIO B50:21/7 NXB XIC B50:21/8 BND OTE B50:13/2 EOR
%   B50:21/1  "Action bunk" %
%   B50:13/2  "pusher_back" %
% Rung: 51 %
% Timeout forward pusher %
SOR XIC B50:21/1 XIC B50:13/1 BST TON T4:37 0.01 700 0 NXB XIC T4:37/DN OTE B50:21/12 BND EOR
%   B50:21/1  "Action bunk" %
%   B50:13/1  "pusher_forward" %
%   T4:37  "TAN-TIMEOUT FORWARD PUSHER" %
% Rung: 52 %
SOR XIO T4:37/EN RES T4:37 EOR
%   T4:37  "TAN-TIMEOUT FORWARD PUSHER" %
% Rung: 53 %
% Timeout back pusher %
SOR XIC B50:21/1 XIC B50:13/2 BST TON T4:38 0.01 700 0 NXB XIC T4:38/DN OTE B50:21/13 BND EOR
%   B50:21/1  "Action bunk" %
%   B50:13/2  "pusher_back" %
%   T4:38  "TAO-TIMEOUT BACK PUSHER" %
% Rung: 54 %
SOR XIO T4:38/EN RES T4:38 EOR
%   T4:38  "TAO-TIMEOUT BACK PUSHER" %
% Rung: 55 %
SOR XIC B50:21/2 XIC B10:100/0 BST OTE B50:14/0 NXB OTE B50:14/1 BND EOR
%   B50:21/2  "Bunk inserted" %
%   B10:100/0  A_STRAP  "A_Strap" %
%   B50:14/0  "X18_1" %
%   B50:14/1  "X19_1" %
% Rung: 56 %
SOR XIC B50:14/0 XIC N11:1/4 OTE N11:1/7 EOR
%   B50:14/0  "X18_1" %

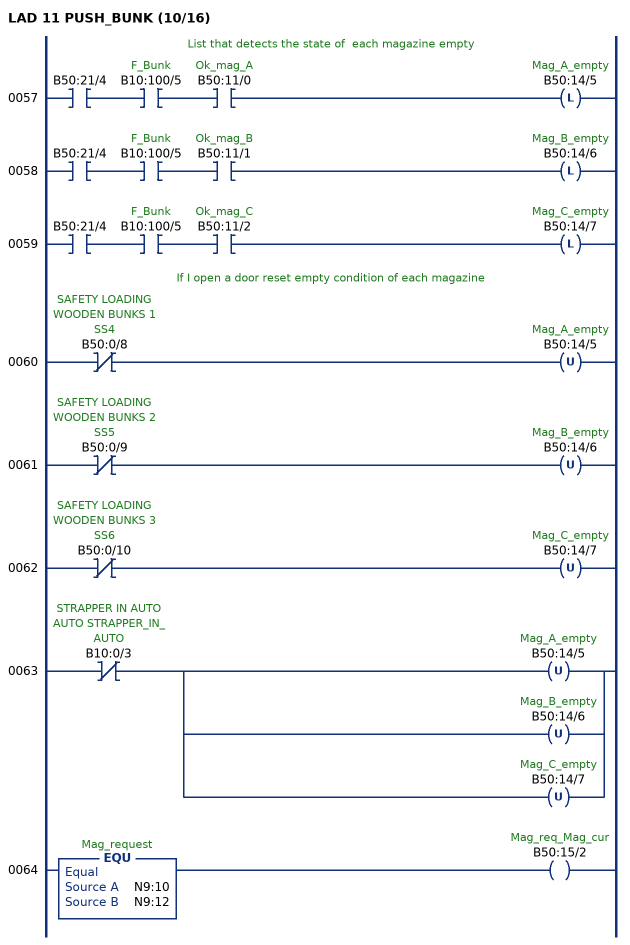
% Rung: 57 %
% List that detects the state of  each magazine empty %
SOR XIC B50:21/4 XIC B10:100/5 XIC B50:11/0 OTL B50:14/5 EOR
%   B10:100/5  "F_Bunk" %
%   B50:11/0  "Ok_mag_A" %
%   B50:14/5  "Mag_A_empty" %
% Rung: 58 %
SOR XIC B50:21/4 XIC B10:100/5 XIC B50:11/1 OTL B50:14/6 EOR
%   B10:100/5  "F_Bunk" %
%   B50:11/1  "Ok_mag_B" %
%   B50:14/6  "Mag_B_empty" %
% Rung: 59 %
SOR XIC B50:21/4 XIC B10:100/5 XIC B50:11/2 OTL B50:14/7 EOR
%   B10:100/5  "F_Bunk" %
%   B50:11/2  "Ok_mag_C" %
%   B50:14/7  "Mag_C_empty" %
% Rung: 60 %
% If I open a door reset empty condition of each magazine %
SOR XIO B50:0/8 OTU B50:14/5 EOR
%   B50:0/8  SS4  "SAFETY LOADING WOODEN BUNKS 1" %
%   B50:14/5  "Mag_A_empty" %
% Rung: 61 %
SOR XIO B50:0/9 OTU B50:14/6 EOR
%   B50:0/9  SS5  "SAFETY LOADING WOODEN BUNKS 2" %
%   B50:14/6  "Mag_B_empty" %
% Rung: 62 %
SOR XIO B50:0/10 OTU B50:14/7 EOR
%   B50:0/10  SS6  "SAFETY LOADING WOODEN BUNKS 3" %
%   B50:14/7  "Mag_C_empty" %
% Rung: 63 %
SOR XIO B10:0/3 BST OTU B50:14/5 NXB BST OTU B50:14/6 NXB OTU B50:14/7 BND BND EOR
%   B10:0/3  STRAPPER_IN_AUTO  "STRAPPER IN AUTO AUTO" %
%   B50:14/5  "Mag_A_empty" %
%   B50:14/6  "Mag_B_empty" %
%   B50:14/7  "Mag_C_empty" %
% Rung: 64 %
SOR EQU N9:10 N9:12 OTE B50:15/2 EOR
%   N9:10  "Mag_request" %
%   N9:12  "Mag_current" %
%   B50:15/2  "Mag_req_Mag_cur" %

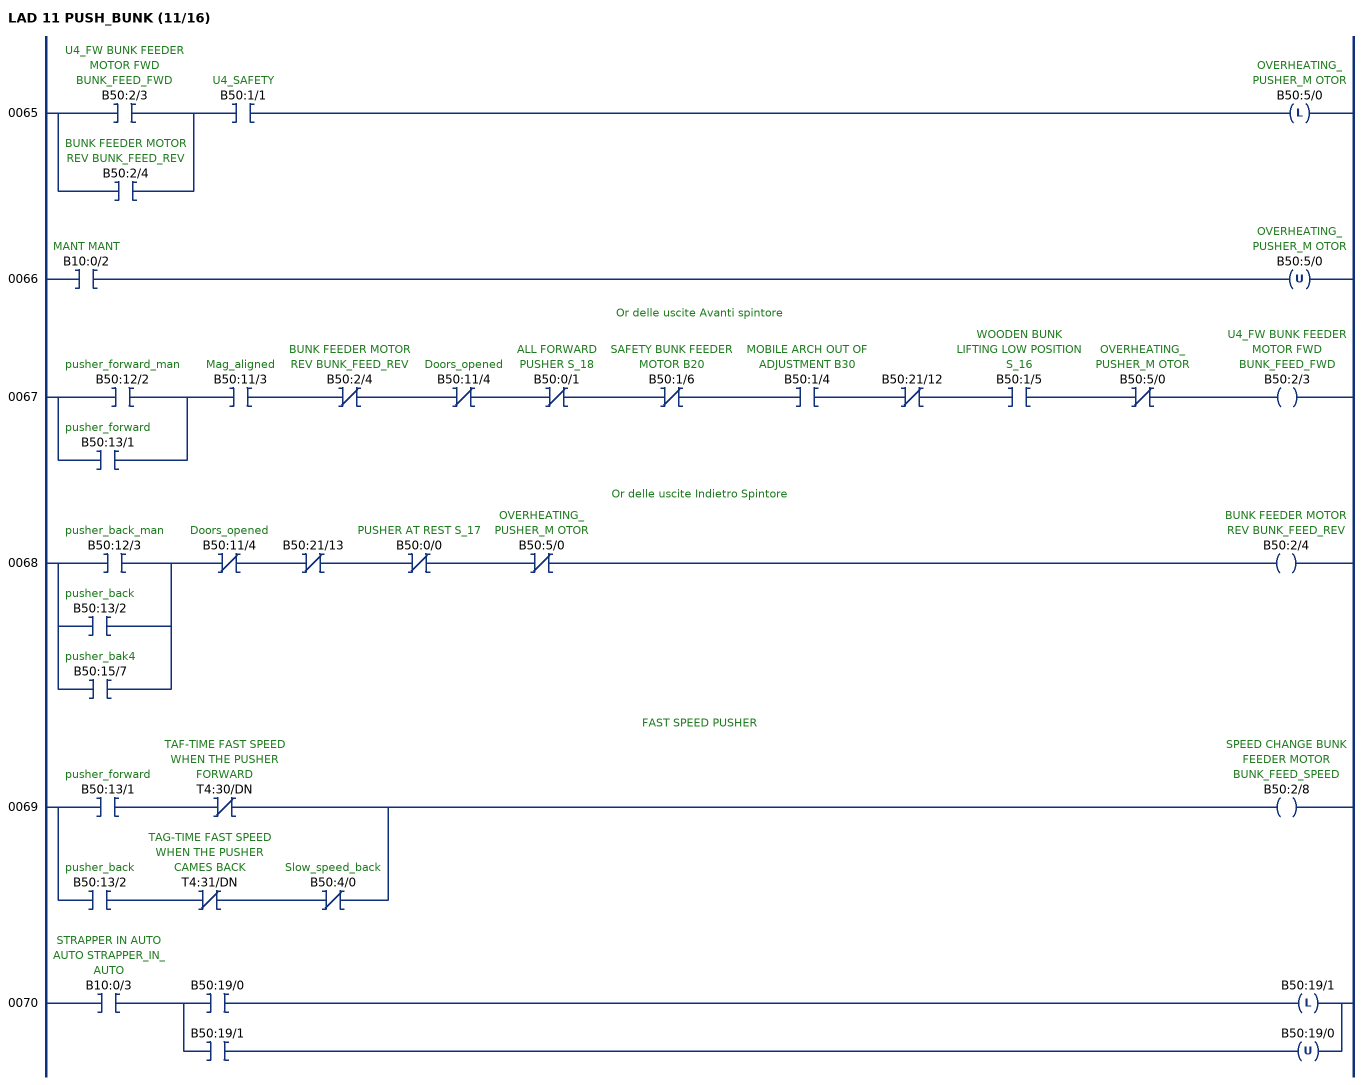
% Rung: 65 %
SOR BST XIC B50:2/3 NXB XIC B50:2/4 BND XIC B50:1/1 OTL B50:5/0 EOR
%   B50:2/3  BUNK_FEED_FWD  "U4_FW BUNK FEEDER MOTOR FWD" %
%   B50:2/4  BUNK_FEED_REV  "BUNK FEEDER MOTOR REV" %
%   B50:1/1  U4_SAFETY %
%   B50:5/0  "OVERHEATING_PUSHER_M OTOR" %
% Rung: 66 %
SOR XIC B10:0/2 OTU B50:5/0 EOR
%   B10:0/2  MANT  "MANT" %
%   B50:5/0  "OVERHEATING_PUSHER_M OTOR" %
% Rung: 67 %
% Or delle uscite Avanti spintore %
SOR BST XIC B50:12/2 NXB XIC B50:13/1 BND XIC B50:11/3 XIO B50:2/4 XIO B50:11/4 XIO B50:0/1 XIO B50:1/6 XIC B50:1/4 XIO B50:21/12 XIC B50:1/5 XIO B50:5/0 OTE B50:2/3 EOR
%   B50:12/2  "pusher_forward_man" %
%   B50:13/1  "pusher_forward" %
%   B50:11/3  "Mag_aligned" %
%   B50:2/4  BUNK_FEED_REV  "BUNK FEEDER MOTOR REV" %
%   B50:11/4  "Doors_opened" %
%   B50:0/1  S_18  "ALL FORWARD PUSHER" %
%   B50:1/6  B20  "SAFETY BUNK FEEDER MOTOR" %
%   B50:1/4  B30  "MOBILE ARCH OUT OF ADJUSTMENT" %
%   B50:1/5  S_16  "WOODEN BUNK LIFTING LOW POSITION" %
%   B50:5/0  "OVERHEATING_PUSHER_M OTOR" %
%   B50:2/3  BUNK_FEED_FWD  "U4_FW BUNK FEEDER MOTOR FWD" %
% Rung: 68 %
% Or delle uscite Indietro Spintore %
SOR BST XIC B50:12/3 NXB BST XIC B50:13/2 NXB XIC B50:15/7 BND BND XIO B50:11/4 XIO B50:21/13 XIO B50:0/0 XIO B50:5/0 OTE B50:2/4 EOR
%   B50:12/3  "pusher_back_man" %
%   B50:13/2  "pusher_back" %
%   B50:15/7  "pusher_bak4" %
%   B50:11/4  "Doors_opened" %
%   B50:0/0  S_17  "PUSHER AT REST" %
%   B50:5/0  "OVERHEATING_PUSHER_M OTOR" %
%   B50:2/4  BUNK_FEED_REV  "BUNK FEEDER MOTOR REV" %
% Rung: 69 %
% FAST SPEED PUSHER %
SOR BST XIC B50:13/1 XIO T4:30/DN NXB XIC B50:13/2 XIO T4:31/DN XIO B50:4/0 BND OTE B50:2/8 EOR
%   B50:13/1  "pusher_forward" %
%   T4:30  "TAF-TIME FAST SPEED WHEN THE PUSHER FORWARD" %
%   B50:13/2  "pusher_back" %
%   T4:31  "TAG-TIME FAST SPEED WHEN THE PUSHER CAMES BACK" %
%   B50:4/0  "Slow_speed_back" %
%   B50:2/8  BUNK_FEED_SPEED  "SPEED CHANGE BUNK FEEDER MOTOR" %
% Rung: 70 %
SOR XIC B10:0/3 BST XIC B50:19/0 OTL B50:19/1 NXB XIC B50:19/1 OTU B50:19/0 BND EOR
%   B10:0/3  STRAPPER_IN_AUTO  "STRAPPER IN AUTO AUTO" %

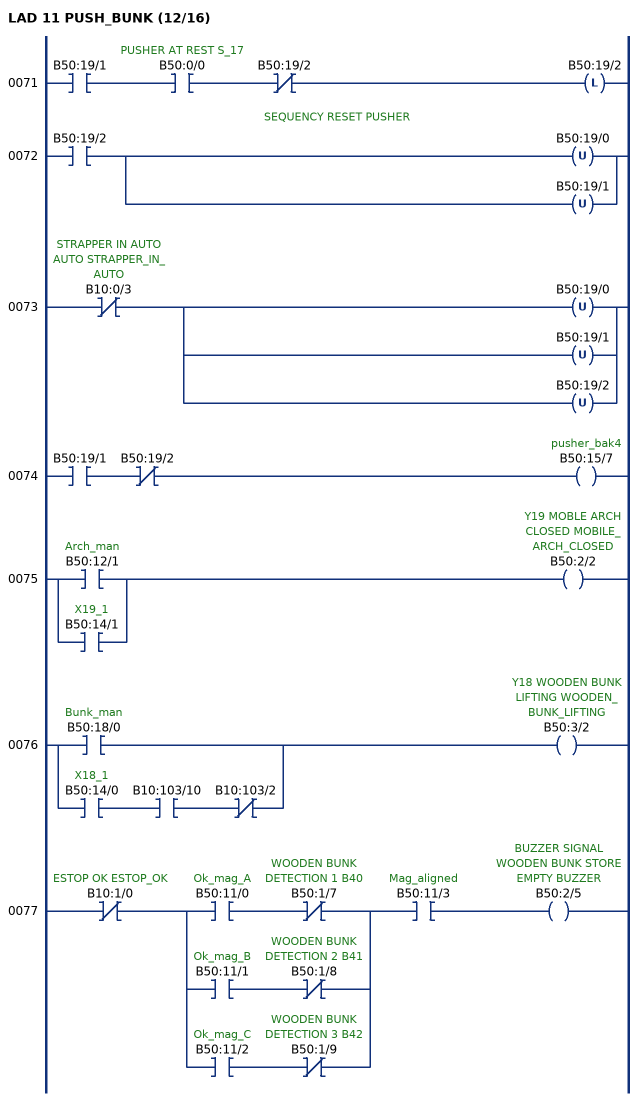
% Rung: 71 %
SOR XIC B50:19/1 XIC B50:0/0 XIO B50:19/2 OTL B50:19/2 EOR
%   B50:0/0  S_17  "PUSHER AT REST" %
% Rung: 72 %
% SEQUENCY RESET PUSHER %
SOR XIC B50:19/2 BST OTU B50:19/0 NXB OTU B50:19/1 BND EOR
% Rung: 73 %
SOR XIO B10:0/3 BST OTU B50:19/0 NXB BST OTU B50:19/1 NXB OTU B50:19/2 BND BND EOR
%   B10:0/3  STRAPPER_IN_AUTO  "STRAPPER IN AUTO AUTO" %
% Rung: 74 %
SOR XIC B50:19/1 XIO B50:19/2 OTE B50:15/7 EOR
%   B50:15/7  "pusher_bak4" %
% Rung: 75 %
SOR BST XIC B50:12/1 NXB XIC B50:14/1 BND OTE B50:2/2 EOR
%   B50:12/1  "Arch_man" %
%   B50:14/1  "X19_1" %
%   B50:2/2  MOBILE_ARCH_CLOSED  "Y19 MOBLE ARCH CLOSED" %
% Rung: 76 %
SOR BST XIC B50:18/0 NXB XIC B50:14/0 XIC B10:103/10 XIO B10:103/2 BND OTE B50:3/2 EOR
%   B50:18/0  "Bunk_man" %
%   B50:14/0  "X18_1" %
%   B50:3/2  WOODEN_BUNK_LIFTING  "Y18 WOODEN BUNK LIFTING" %
% Rung: 77 %
SOR XIO B10:1/0 BST XIC B50:11/0 XIO B50:1/7 NXB BST XIC B50:11/1 XIO B50:1/8 NXB XIC B50:11/2 XIO B50:1/9 BND BND XIC B50:11/3 OTE B50:2/5 EOR
%   B10:1/0  ESTOP_OK  "ESTOP OK" %
%   B50:11/0  "Ok_mag_A" %
%   B50:1/7  B40  "WOODEN BUNK DETECTION 1" %
%   B50:11/1  "Ok_mag_B" %
%   B50:1/8  B41  "WOODEN BUNK DETECTION 2" %
%   B50:11/2  "Ok_mag_C" %
%   B50:1/9  B42  "WOODEN BUNK DETECTION 3" %
%   B50:11/3  "Mag_aligned" %
%   B50:2/5  BUZZER  "BUZZER SIGNAL WOODEN BUNK STORE EMPTY" %

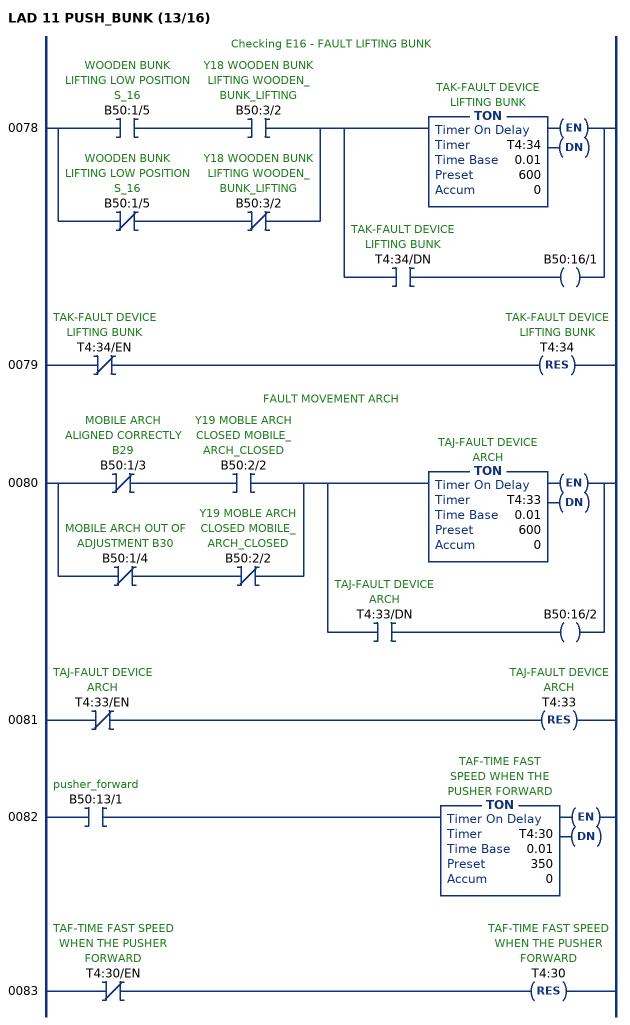
% Rung: 78 %
% Checking E16 - FAULT LIFTING BUNK %
SOR BST XIC B50:1/5 XIC B50:3/2 NXB XIO B50:1/5 XIO B50:3/2 BND BST TON T4:34 0.01 600 0 NXB XIC T4:34/DN OTE B50:16/1 BND EOR
%   B50:1/5  S_16  "WOODEN BUNK LIFTING LOW POSITION" %
%   B50:3/2  WOODEN_BUNK_LIFTING  "Y18 WOODEN BUNK LIFTING" %
%   T4:34  "TAK-FAULT DEVICE LIFTING BUNK" %
% Rung: 79 %
SOR XIO T4:34/EN RES T4:34 EOR
%   T4:34  "TAK-FAULT DEVICE LIFTING BUNK" %
% Rung: 80 %
% FAULT MOVEMENT ARCH %
SOR BST XIO B50:1/3 XIC B50:2/2 NXB XIO B50:1/4 XIO B50:2/2 BND BST TON T4:33 0.01 600 0 NXB XIC T4:33/DN OTE B50:16/2 BND EOR
%   B50:1/3  B29  "MOBILE ARCH ALIGNED CORRECTLY" %
%   B50:2/2  MOBILE_ARCH_CLOSED  "Y19 MOBLE ARCH CLOSED" %
%   B50:1/4  B30  "MOBILE ARCH OUT OF ADJUSTMENT" %
%   T4:33  "TAJ-FAULT DEVICE ARCH" %
% Rung: 81 %
SOR XIO T4:33/EN RES T4:33 EOR
%   T4:33  "TAJ-FAULT DEVICE ARCH" %
% Rung: 82 %
SOR XIC B50:13/1 TON T4:30 0.01 350 0 EOR
%   B50:13/1  "pusher_forward" %
%   T4:30  "TAF-TIME FAST SPEED WHEN THE PUSHER FORWARD" %
% Rung: 83 %
SOR XIO T4:30/EN RES T4:30 EOR
%   T4:30  "TAF-TIME FAST SPEED WHEN THE PUSHER FORWARD" %

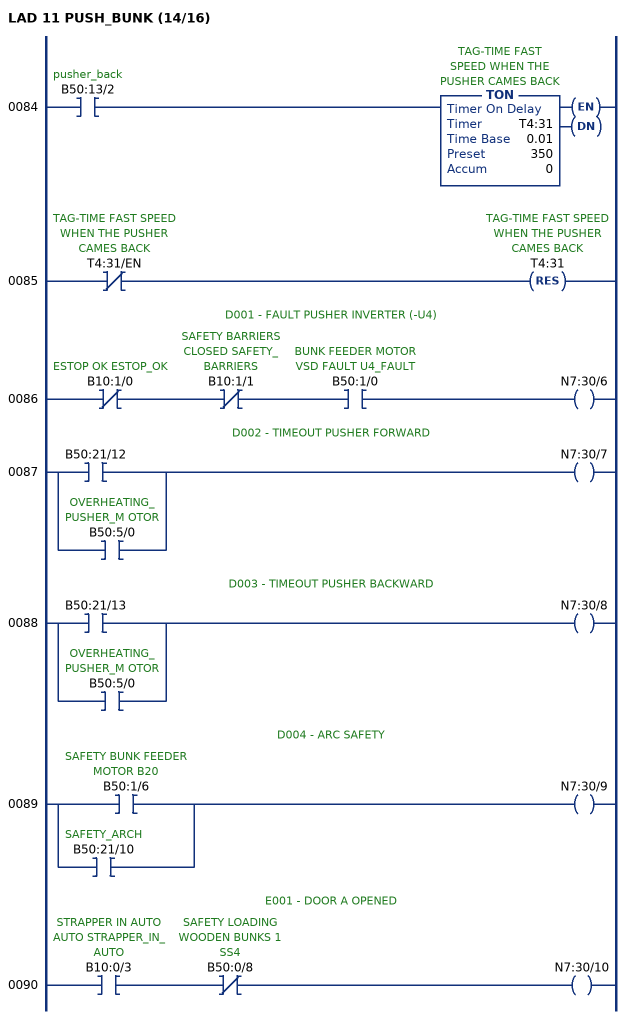
% Rung: 84 %
SOR XIC B50:13/2 TON T4:31 0.01 350 0 EOR
%   B50:13/2  "pusher_back" %
%   T4:31  "TAG-TIME FAST SPEED WHEN THE PUSHER CAMES BACK" %
% Rung: 85 %
SOR XIO T4:31/EN RES T4:31 EOR
%   T4:31  "TAG-TIME FAST SPEED WHEN THE PUSHER CAMES BACK" %
% Rung: 86 %
% D001 - FAULT PUSHER INVERTER (-U4) %
SOR XIO B10:1/0 XIO B10:1/1 XIC B50:1/0 OTE N7:30/6 EOR
%   B10:1/0  ESTOP_OK  "ESTOP OK" %
%   B10:1/1  SAFETY_BARRIERS  "SAFETY BARRIERS CLOSED" %
%   B50:1/0  U4_FAULT  "BUNK FEEDER MOTOR VSD FAULT" %
% Rung: 87 %
% D002 - TIMEOUT PUSHER FORWARD %
SOR BST XIC B50:21/12 NXB XIC B50:5/0 BND OTE N7:30/7 EOR
%   B50:5/0  "OVERHEATING_PUSHER_M OTOR" %
% Rung: 88 %
% D003 - TIMEOUT PUSHER BACKWARD %
SOR BST XIC B50:21/13 NXB XIC B50:5/0 BND OTE N7:30/8 EOR
%   B50:5/0  "OVERHEATING_PUSHER_M OTOR" %
% Rung: 89 %
% D004 - ARC SAFETY %
SOR BST XIC B50:1/6 NXB XIC B50:21/10 BND OTE N7:30/9 EOR
%   B50:1/6  B20  "SAFETY BUNK FEEDER MOTOR" %
%   B50:21/10  "SAFETY_ARCH" %
% Rung: 90 %
% E001 - DOOR A OPENED %
SOR XIC B10:0/3 XIO B50:0/8 OTE N7:30/10 EOR
%   B10:0/3  STRAPPER_IN_AUTO  "STRAPPER IN AUTO AUTO" %
%   B50:0/8  SS4  "SAFETY LOADING WOODEN BUNKS 1" %

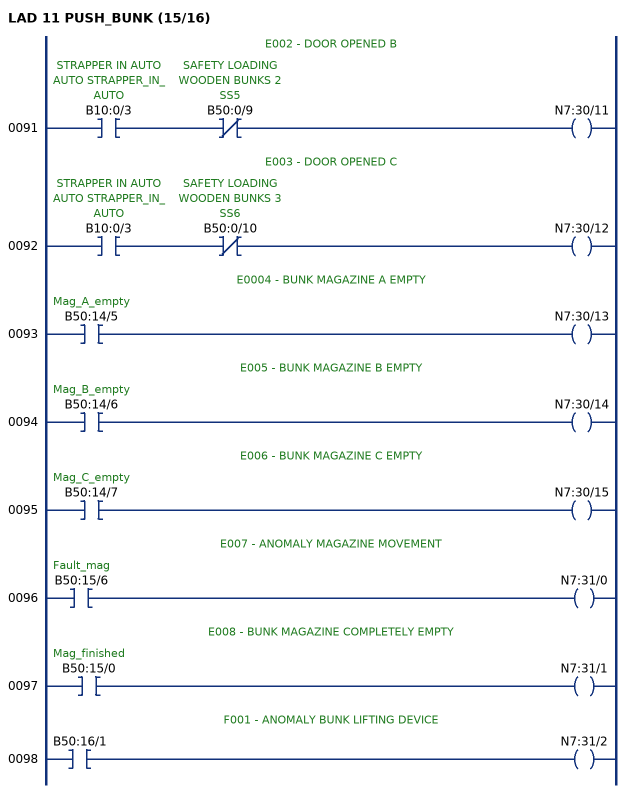
% Rung: 91 %
% E002 - DOOR OPENED B %
SOR XIC B10:0/3 XIO B50:0/9 OTE N7:30/11 EOR
%   B10:0/3  STRAPPER_IN_AUTO  "STRAPPER IN AUTO AUTO" %
%   B50:0/9  SS5  "SAFETY LOADING WOODEN BUNKS 2" %
% Rung: 92 %
% E003 - DOOR OPENED C %
SOR XIC B10:0/3 XIO B50:0/10 OTE N7:30/12 EOR
%   B10:0/3  STRAPPER_IN_AUTO  "STRAPPER IN AUTO AUTO" %
%   B50:0/10  SS6  "SAFETY LOADING WOODEN BUNKS 3" %
% Rung: 93 %
% E0004 - BUNK MAGAZINE A EMPTY %
SOR XIC B50:14/5 OTE N7:30/13 EOR
%   B50:14/5  "Mag_A_empty" %
% Rung: 94 %
% E005 - BUNK MAGAZINE B EMPTY %
SOR XIC B50:14/6 OTE N7:30/14 EOR
%   B50:14/6  "Mag_B_empty" %
% Rung: 95 %
% E006 - BUNK MAGAZINE C EMPTY %
SOR XIC B50:14/7 OTE N7:30/15 EOR
%   B50:14/7  "Mag_C_empty" %
% Rung: 96 %
% E007 - ANOMALY MAGAZINE MOVEMENT %
SOR XIC B50:15/6 OTE N7:31/0 EOR
%   B50:15/6  "Fault_mag" %
% Rung: 97 %
% E008 - BUNK MAGAZINE COMPLETELY EMPTY %
SOR XIC B50:15/0 OTE N7:31/1 EOR
%   B50:15/0  "Mag_finished" %
% Rung: 98 %
% F001 - ANOMALY BUNK LIFTING DEVICE %
SOR XIC B50:16/1 OTE N7:31/2 EOR

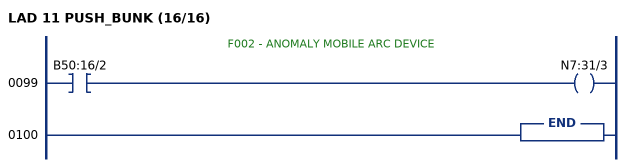
% Rung: 99 %
% F002 - ANOMALY MOBILE ARC DEVICE %
SOR XIC B50:16/2 OTE N7:31/3 EOR
% Rung: 100 %
SOR END EOR

LADDER 12 "CHECKING"
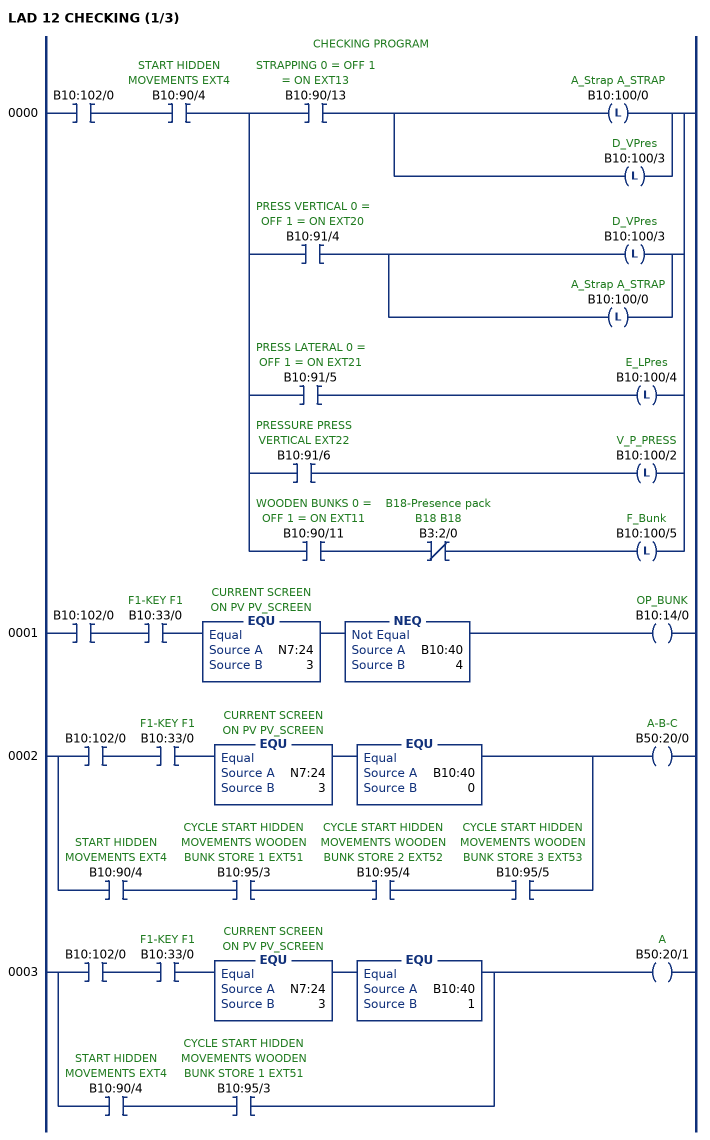
% Rung: 0 %
% CHECKING PROGRAM %
SOR XIC B10:102/0 XIC B10:90/4 BST BST XIC B10:90/13 BST OTL B10:100/0 NXB OTL B10:100/3 BND NXB BST XIC B10:91/4 BST OTL B10:100/3 NXB OTL B10:100/0 BND NXB BST XIC B10:91/5 OTL B10:100/4 NXB XIC B10:91/6 OTL B10:100/2 BND BND BND NXB XIC B10:90/11 XIO B3:2/0 OTL B10:100/5 BND EOR
%   B10:90/4  EXT4  "START HIDDEN MOVEMENTS" %
%   B10:90/13  EXT13  "STRAPPING 0 = OFF 1 = ON" %
%   B10:100/0  A_STRAP  "A_Strap" %
%   B10:100/3  "D_VPres" %
%   B10:91/4  EXT20  "PRESS VERTICAL 0 = OFF 1 = ON" %
%   B10:91/5  EXT21  "PRESS LATERAL 0 = OFF 1 = ON" %
%   B10:100/4  "E_LPres" %
%   B10:91/6  EXT22  "PRESSURE PRESS VERTICAL" %
%   B10:100/2  "V_P_PRESS" %
%   B10:90/11  EXT11  "WOODEN BUNKS 0 = OFF 1 = ON" %
%   B3:2/0  B18  "B18-Presence pack B18" %
%   B10:100/5  "F_Bunk" %
% Rung: 1 %
SOR XIC B10:102/0 XIC B10:33/0 EQU N7:24 3 NEQ B10:40 4 OTE B10:14/0 EOR
%   B10:33/0  F1  "F1-KEY" %
%   N7:24  PV_SCREEN  "CURRENT SCREEN ON PV" %
%   B10:14/0  "OP_BUNK" %
% Rung: 2 %
SOR BST XIC B10:102/0 XIC B10:33/0 EQU N7:24 3 EQU B10:40 0 NXB XIC B10:90/4 XIC B10:95/3 XIC B10:95/4 XIC B10:95/5 BND OTE B50:20/0 EOR
%   B10:33/0  F1  "F1-KEY" %
%   N7:24  PV_SCREEN  "CURRENT SCREEN ON PV" %
%   B10:90/4  EXT4  "START HIDDEN MOVEMENTS" %
%   B10:95/3  EXT51  "CYCLE START HIDDEN MOVEMENTS WOODEN BUNK STORE 1" %
%   B10:95/4  EXT52  "CYCLE START HIDDEN MOVEMENTS WOODEN BUNK STORE 2" %
%   B10:95/5  EXT53  "CYCLE START HIDDEN MOVEMENTS WOODEN BUNK STORE 3" %
%   B50:20/0  "A-B-C" %
% Rung: 3 %
SOR BST XIC B10:102/0 XIC B10:33/0 EQU N7:24 3 EQU B10:40 1 NXB XIC B10:90/4 XIC B10:95/3 BND OTE B50:20/1 EOR
%   B10:33/0  F1  "F1-KEY" %
%   N7:24  PV_SCREEN  "CURRENT SCREEN ON PV" %
%   B10:90/4  EXT4  "START HIDDEN MOVEMENTS" %
%   B10:95/3  EXT51  "CYCLE START HIDDEN MOVEMENTS WOODEN BUNK STORE 1" %
%   B50:20/1  "A" %

